FUNCTION_BLOCK FB_GeoEllipsoid_Test EXTENDS FB_TestSuite
VAR_INPUT
END_VAR
VAR_OUTPUT
END_VAR
VAR
END_VAR

WhenReferenceConstantExpectItExists();
WhenGetCartesianExpectValue();
WhenGetGeodeticExpectValue();
WhenTransformEnuAltExpectValue();
WhenTransformEnulatLonExpectValue();

METHOD PRIVATE WhenGetCartesianExpectValue
VAR_INPUT
	
END_VAR
VAR
	PX : GeoPosition;
	PY : GeoPosition;
	PZ : GeoPosition;
	VX : Vector3;
	VY : Vector3;
	VZ : Vector3;
END_VAR
TEST('WhenGetCartesianExpectValue');

// @TEST-RUN
PX.SetFromComponentsDeg(0,0,1);
PY.SetFromComponentsDeg(0,90,1);
PZ.SetFromComponentsDeg(90,0,1);
VX := GeoEllipsoids.WGS84.GetCartesianFromGeodetic(PX);
VY := GeoEllipsoids.WGS84.GetCartesianFromGeodetic(PY);
VZ := GeoEllipsoids.WGS84.GetCartesianFromGeodetic(PZ);

// @TEST-ASSERT
AssertTrue(VX.X = GeoEllipsoids.WGS84.SemiMajorAxis+1, 'X axis check does not work');
AssertTrue(VY.Y = GeoEllipsoids.WGS84.SemiMajorAxis+1, 'Y axis check does not work');
AssertTrue(VZ.Z = (1-GeoEllipsoids.WGS84.Flattening)*GeoEllipsoids.WGS84.SemiMajorAxis +1, 'Z axis check does not work');


TEST_FINISHED();
END_METHOD

METHOD PRIVATE WhenGetGeodeticExpectValue
VAR_INPUT
	
END_VAR
VAR
	PX : GeoPosition;
	PY : GeoPosition;
	PZ : GeoPosition;
	PXYZ : GeoPosition;
	VX : Vector3;
	VXb : Vector3;
	VY : Vector3;
	VZ : Vector3;
	VXYZ : Vector3;
	PX2 : GeoPosition;
	PX2b : GeoPosition;
	PY2 : GeoPosition;
	PZ2 : GeoPosition;
	PXYZ2 : GeoPosition;
END_VAR
TEST('WhenGetGeodeticExpectValue');

// @TEST-RUN
PX.SetFromComponentsDeg(0,0,1);
PY.SetFromComponentsDeg(0,90,1);
PZ.SetFromComponentsDeg(90,0,1);
PXYZ.SetFromComponentsDeg(45,45,1000);
VX := GeoEllipsoids.WGS84.GetCartesianFromGeodetic(PX);
VXb := GeoEllipsoids.WGS84.GetCartesianFromGeodetic(PX);
VXb.Z := VXb.Z - 1;//just south of equator
VY := GeoEllipsoids.WGS84.GetCartesianFromGeodetic(PY);
VZ := GeoEllipsoids.WGS84.GetCartesianFromGeodetic(PZ);
VXYZ := GeoEllipsoids.WGS84.GetCartesianFromGeodetic(PXYZ);
PX2 := GeoEllipsoids.WGS84.GetGeodeticFromCartesian(VX);
PX2b := GeoEllipsoids.WGS84.GetGeodeticFromCartesian(VXb);
PY2 := GeoEllipsoids.WGS84.GetGeodeticFromCartesian(VY);
PZ2 := GeoEllipsoids.WGS84.GetGeodeticFromCartesian(VZ);
PXYZ2 := GeoEllipsoids.WGS84.GetGeodeticFromCartesian(VXYZ);

// @TEST-ASSERT
AssertTrue(PX.IsNearlyEqual(PX2,1E-6), 'X axis check does not work');
AssertTrue(PY.IsNearlyEqual(PY2,1E-6), 'Y axis check does not work');
AssertTrue(PZ.IsNearlyEqual(PZ2,1E-6), 'Z axis check does not work');
AssertTrue(PXYZ.IsNearlyEqual(PXYZ2,1E-6), 'Compound axis check does not work');

AssertTrue(PX2b.LatitudeRad < 0, 'Small latitude perturbation does not work');


TEST_FINISHED();
END_METHOD

METHOD PRIVATE WhenReferenceConstantExpectItExists
VAR_INPUT
END_VAR
VAR
	WGS84 : REFERENCE TO GeoEllipsoid;
END_VAR
TEST('WhenReferenceConstantExpectItExists');

// @TEST-RUN
WGS84 REF=  GeoEllipsoids.WGS84;

// @TEST-ASSERT
AssertTrue(WGS84.SemiMajorAxis = 6378137, 'semi major axis not right');
AssertTrue(WGS84.Flattening = 1.0 / 298.257223563, 'flattening not right');

TEST_FINISHED();
END_METHOD

METHOD PRIVATE WhenTransformEnuAltExpectValue
VAR_INPUT
	
END_VAR
VAR
	Psurf : GeoPosition;
	Palt : GeoPosition;
	Vsurf : Vector3;
	Valt : Vector3;
	Valt_surf : Vector3;
	Hsurf : HMatrix;
	Valt2 : Vector3;
END_VAR
TEST('WhenTransformEnuAltExpectValue');

// @TEST-RUN
Psurf.SetFromComponentsDeg(0,0,0);
Palt.SetFromComponentsDeg(PSurf.LatitudeDeg,PSurf.LongitudeDeg,1000);
Valt_surf.SetFromComponents(0,0,Palt.Elevation);

Vsurf := GeoEllipsoids.WGS84.GetCartesianFromGeodetic(Psurf);
Valt := GeoEllipsoids.WGS84.GetCartesianFromGeodetic(Palt);
Hsurf := GeoEllipsoids.WGS84.GetTangentEnuTransform(Psurf);
Valt2 := Hsurf.GetTransformedVector3(Valt_surf);

// @TEST-ASSERT
AssertTrue(Valt.IsNearlyEqual(Valt2,1E-6), 'transformation did not work');


TEST_FINISHED();
END_METHOD

METHOD PRIVATE WhenTransformEnuLatLonExpectValue
VAR_INPUT
	
END_VAR
VAR
	Psurf : GeoPosition;
	Palt : GeoPosition;
	Vsurf : Vector3;
	Valt : Vector3;
	Valt_surf : Vector3;
	Hsurf : HMatrix;
	Valt2 : Vector3;
END_VAR
TEST('WhenTransformEnuLatLonExpectValue');

// @TEST-RUN
Psurf.SetFromComponentsDeg(10,10,0);
Palt.SetFromComponentsDeg(PSurf.LatitudeDeg,PSurf.LongitudeDeg,1000);
Valt_surf.SetFromComponents(0,0,Palt.Elevation);

Vsurf := GeoEllipsoids.WGS84.GetCartesianFromGeodetic(Psurf);
Valt := GeoEllipsoids.WGS84.GetCartesianFromGeodetic(Palt);
Hsurf := GeoEllipsoids.WGS84.GetTangentEnuTransform(Psurf);
Valt2 := Hsurf.GetTransformedVector3(Valt_surf);

// @TEST-ASSERT
AssertTrue(Valt.IsNearlyEqual(Valt2,1E-6), 'transformation did not work');


TEST_FINISHED();
END_METHOD

END_FUNCTION_BLOCK

(* stored: Version 1.1.0.1, ProductVersion 3.1.4024.9
   POU FB_GeoEllipsoid_Test: Id {2c826b29-42af-412b-b9f6-6027132ceddb}, SpecialFunc None
   Method WhenGetCartesianExpectValue: Id {b09fafe1-6b82-4288-9315-605ef0b78999}
   Method WhenGetGeodeticExpectValue: Id {05fd3b87-4737-431f-a99d-4d1552991f37}
   Method WhenReferenceConstantExpectItExists: Id {4b7e9965-97b5-43a8-81ef-de5a019d91ff}
   Method WhenTransformEnuAltExpectValue: Id {b7da807a-920e-457d-8e20-a816d1108f30}
   Method WhenTransformEnuLatLonExpectValue: Id {84ac00c5-743a-4fbd-b395-53e78229cb25} *)
